// Mitsubishi GX Works2 project: test_in_out_fx1nc   PLC: FX1N/FX1NC

PROGRAM MAIN
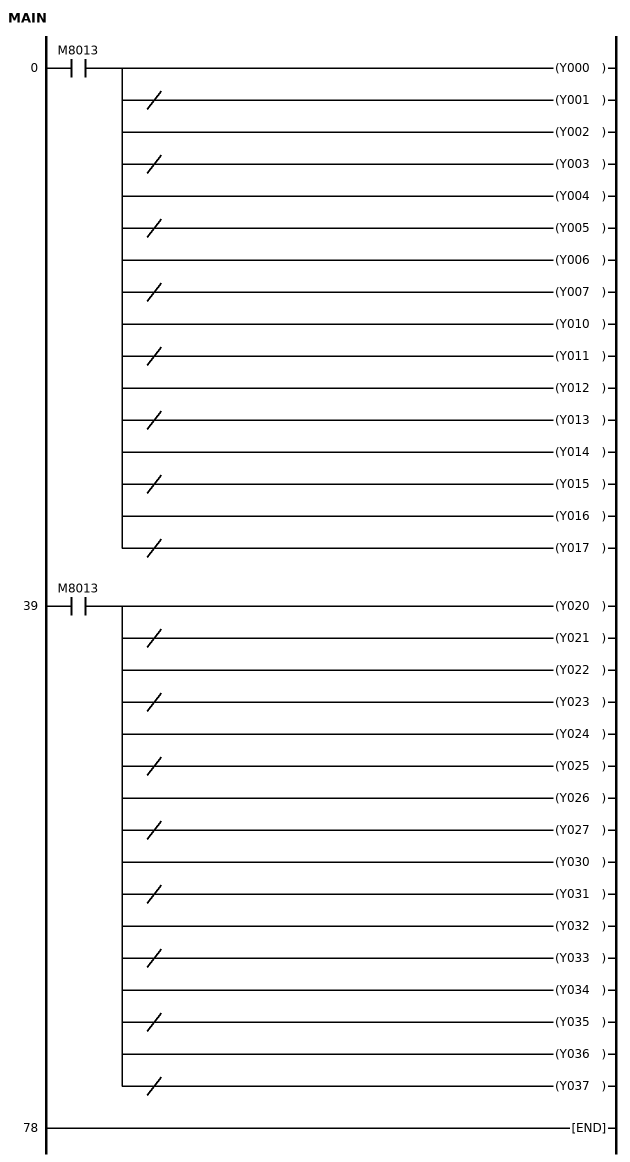
0     LD      M8013
      OUT     Y000
      MPS
      INV
      OUT     Y001
      MPP
      OUT     Y002
      MPS
      INV
      OUT     Y003
      MPP
      OUT     Y004
      MPS
      INV
      OUT     Y005
      MPP
      OUT     Y006
      MPS
      INV
      OUT     Y007
      MPP
      OUT     Y010
      MPS
      INV
      OUT     Y011
      MPP
      OUT     Y012
      MPS
      INV
      OUT     Y013
      MPP
      OUT     Y014
      MPS
      INV
      OUT     Y015
      MPP
      OUT     Y016
      INV
      OUT     Y017
39    LD      M8013
      OUT     Y020
      MPS
      INV
      OUT     Y021
      MPP
      OUT     Y022
      MPS
      INV
      OUT     Y023
      MPP
      OUT     Y024
      MPS
      INV
      OUT     Y025
      MPP
      OUT     Y026
      MPS
      INV
      OUT     Y027
      MPP
      OUT     Y030
      MPS
      INV
      OUT     Y031
      MPP
      OUT     Y032
      MPS
      INV
      OUT     Y033
      MPP
      OUT     Y034
      MPS
      INV
      OUT     Y035
      MPP
      OUT     Y036
      INV
      OUT     Y037
78    END
END_PROGRAM
